{attribute 'GeneratedUsingTerminal: EL3052-0000-0016'}
{attribute addProperty BoxType "EL3052-0000-0016"}
{attribute addProperty Id "AI_Standard_Channel_1AT %I*AI_Standard_Channel_EA9DF21E9AI_Standard_Channel_2AT %I*AI_Standard_Channel_EA9DF21E9WcStateAT %I*WcState_9091E0EB2InfoDataAT %I*InfoData_94A18F5E2"}
{attribute addProperty CRC "3858422835"}
{attribute addProperty Size "22"}
TYPE EL3052_E5FADC33 EXTENDS EtcSlaveTerminalBase_947E5A46 :
STRUCT
	{attribute addProperty Name "AI_Standard_Channel_1"}
	AI_Standard_Channel_1 : AI_Standard_Channel_EA9DF21E;
	{attribute addProperty Name "AI_Standard_Channel_2"}
	AI_Standard_Channel_2 : AI_Standard_Channel_EA9DF21E;
	{attribute addProperty Name "WcState"}
	WcState : WcState_9091E0EB;
	{attribute addProperty Name "InfoData"}
	InfoData : InfoData_94A18F5E;
END_STRUCT
END_TYPE

(* stored: Version 1.2.0.0, ProductVersion 3.1.4024.9
   DUT EL3052_E5FADC33: Id {0f370913-af3d-43a9-92d7-7ceb30b54643} *)
